(* IEC 61131-3 sources: brOscatLib/oscatBasic_tests/test_SENSOR_INT, 3 files *)

(* ---- actions.st ---- *)
ACTION TEST_CASE_1_SETUP :
    IF vTestCases[0].state = ut_SETUP THEN
    	(*Setup the test case information*)
    	vTestCases[0].id := 1;
    	vTestCases[0].desc[0] := '';
        vTestCases[0].desc[1] := '';

    	(*Setup needed variables*)

    END_IF
END_ACTION
ACTION TEST_CASE_1_EXEC :
    IF vTestCases[0].state = ut_RUNNING THEN
    	(*Run the test case*)
    		vTestCases[0].state := ut_FAILED;
    		vTestCases[0].msg := 'Test case not implemented -> FAIL';
    END_IF
END_ACTION
ACTION TEST_CASE_2_SETUP :
    IF vTestCases[1].state = ut_SETUP THEN
    	(*Setup the test case information*)
    	vTestCases[1].id := 2;
    	vTestCases[1].desc[0] := '';
        vTestCases[1].desc[1] := '';
    	vTestCases[1].desc[2] := '';

    	(*Setup needed variables*)
    END_IF
END_ACTION
ACTION TEST_CASE_2_EXEC :
    IF vTestCases[1].state = ut_RUNNING THEN
    	(*Run the test case*)
    		vTestCases[1].state := ut_FAILED;
    		vTestCases[1].msg := 'Test case not implemented -> FAIL';
    END_IF
END_ACTION

(* ---- LocalVariables.var ---- *)
VAR
    vTestCases : ARRAY[0..20] OF utTestCase; (*Definition of all test cases for this POU*)
    testRunner : utTestSuite; (*Test Suite fb instance to run the tests*)
    vRunAll : BOOL; (*Manual command to run all tests for this POU*)
    vResetAll : BOOL; (*Manual command to reset all tests for this POU*)
END_VAR

(* ---- main.st ---- *)
PROGRAM _CYCLIC
    (*This PRG tests the functionality of the SENSOR_INT as described in the function description
	http://www.oscat.de/images/OSCATBasic/oscat_basic333_en.pdf#page=324*)
    (*Run the test cases*)
    TEST_CASE_1_SETUP;
    TEST_CASE_1_EXEC;

    TEST_CASE_2_SETUP;
    TEST_CASE_2_EXEC;

    (*Instantiate the test runner*)
    testRunner(
    	Id := 104,
    	Name := 'SENSOR_INT',
        RunTests := gRunAll OR vRunAll,
    	ResetTests := gResetAll OR vResetAll,
    	TestCases:=vTestCases);

    (*Report the results to the collection global*)
    gResults[testRunner.Id] := testRunner.Summary;
END_PROGRAM
